FUNCTION TryConvert_INT_TO_ULINT : BOOL
VAR_INPUT
	in : INT;
	out : REFERENCE TO ULINT;
END_VAR

IF in < DatatypeLimits.MIN_VALUE_OF_INT_WHICH_CAN_BE_HELD_IN_A_ULINT THEN
	RETURN;
END_IF

out := INT_TO_ULINT(in);
TryConvert_INT_TO_ULINT := TRUE;

END_FUNCTION

(* stored: Version 1.1.0.1, ProductVersion 3.1.4024.12
   POU TryConvert_INT_TO_ULINT: Id {f907ed29-fd89-4549-ae91-a055e6fabdc2}, SpecialFunc None *)
